FUNCTION_BLOCK FB_setupAdjustDetect
VAR_INPUT
END_VAR
VAR_OUTPUT
END_VAR
VAR
	m_manualAdjustOnCounts :INT :=0;
	m_adjustOnCountThres :INT :=50;
END_VAR

METHOD run : BOOL
VAR_INPUT
	IOValue :UDINT;
END_VAR

VAR_OUTPUT
	
END_VAR
// manuel adjust io is 5th bit 
IF 16=(IOValue AND 10#16) THEN
	m_manualAdjustOnCounts :=MIN(m_manualAdjustOnCounts +1,m_adjustOnCountThres);
ELSE
	m_manualAdjustOnCounts :=0;
END_IF

run := m_manualAdjustOnCounts >= m_adjustOnCountThres;
END_METHOD

END_FUNCTION_BLOCK

(* stored: Version 1.1.0.1, ProductVersion 3.1.4024.11
   POU FB_setupAdjustDetect: Id {c0770542-a14f-401c-951e-b289373a905f}, SpecialFunc None
   Method run: Id {9417d02d-486a-427f-b657-d20113e6f4a0} *)
